Staubli VAL3: start.pgx

public program start()
begin
  //所有的IO动作都要写入log文件中
  //信号一般作为脉冲信号来处理
  //



  call Init()

  while true


    call Digtal2Analog()
    delay(0)
  endWhile
end
